FUNCTION_BLOCK Test_TStreamAddReadArgType EXTENDS T_UnitTestBase
VAR
    Stream : T_Stream(StreamLength := 2);
END_VAR

Stream.Init(2);

Stream.SetNextArgTypeId(E_ArgTypeId.Type_LINT);

Assertion.AssertEquals_UDINT(Expected     := 2,
                             Actual       := Stream.Position,
                             VariableName := 'Stream.Position');

Stream.Seek(0);

Assertion.AssertEquals_INT(Expected     := E_ArgTypeId.Type_LINT,
                           Actual       := Stream.GetNextArgTypeId(),
                           VariableName := 'Stream.GetNextArgTypeId()');

Assertion.AssertEquals_UDINT(Expected     := 2,
                             Actual       := Stream.Position,
                             VariableName := 'Stream.Position');

TestFinished();

END_FUNCTION_BLOCK

(* stored: Version 1.1.0.1, ProductVersion 3.1.4024.6
   POU Test_TStreamAddReadArgType: Id {1360d495-e9de-41ec-9150-13951a2d63ad}, SpecialFunc None *)
